FUNCTION_BLOCK DigitalInput EXTENDS BaseIO
VAR_INPUT
	ProcessValue: BOOL;
	Override: BOOL;
	OverrideValue: BOOL;
	Inverted: bool;
END_VAR
VAR_OUTPUT
	Value: BOOL;
END_VAR
VAR
	InitDone: BOOL;
	TempValue: bool;
END_VAR
VAR PERSISTENT
	IsInverted: BOOL;
	SavedOverride: BOOL;
	SavedOverrideValue: BOOL;
END_VAR

SUPER^();
IF NOT InitDone THEN
	InitDone := TRUE;
	OverrideValue := SavedOverrideValue;
	Override := SavedOverride;	
END_IF
IsInverted := Inverted;

SavedOverride := Override;
SavedOverrideValue := OverrideValue;

IF NOT Override THEN
	TempValue := ProcessValue;
ELSE
	TempValue := OverrideValue;	
END_IF

IF IsInverted THEN
	TempValue := NOT TempValue;
END_IF

Value := TempValue;

END_FUNCTION_BLOCK

(* stored: Version 1.1.0.1, ProductVersion 3.1.4024.5
   POU DigitalInput: Id {3f6e813c-0865-421b-aa64-955fd14f7081}, SpecialFunc None *)
